(* CODESYS project SPT_XPlanar.library
   Company: Beckhoff Automation LLC
   DefaultNamespace: SPT_XPlanar
   Version: 3.2.0
   Placeholder: SPT_XPlanar
   Title: SPT_XPlanar

Project tree, tasks and I/O mapping:
  libraries: SPT Base Types, * (Beckhoff Automation LLC); SPT Event Logger, * (Beckhoff Automation LLC); SPT Tracing, * (Beckhoff Automation LLC); SPT Utilities, * (Beckhoff Automation LLC); Tc2_Math, * (Beckhoff Automation GmbH); Tc2_Standard, * (Beckhoff Automation GmbH); Tc2_System, * (Beckhoff Automation GmbH); Tc2_Utilities, * (Beckhoff Automation GmbH); Tc3_EventLogger, * (Beckhoff Automation GmbH); Tc3_Mc3PlanarMotion, * (Beckhoff Automation GmbH); Tc3_Module, * (Beckhoff Automation GmbH); Tc3_Physics, * (Beckhoff Automation GmbH); Tc3_XPlanarStandard, * (Beckhoff Automation GmbH); Tc3_XPlanarUtility, * (Beckhoff Automation GmbH & Co. KG)
  DUT/
    HMI/
      data type ST_Xplanar_Command
      data type ST_Xplanar_Config
      data type ST_Xplanar_HMI
      data type ST_Xplanar_Status
  Mover/
    DUTs/
      HMI/
        data type ST_Mover_HMI
        data type ST_MoverCommand_HMI
        data type ST_MoverConfig_HMI
        data type ST_MoverStatus_HMI
      data type ST_MoveDynamics
    function block FB_XPlanarMover [ST]: ClearCmd, Destination, Error, ErrorID, ErrorInfo, InStation, MoveDynamics, MoverBTN, MoverIndex, MoverType, std, TrackId, Disable, Enable, FreeMove, Index, JoinTrack, LeaveTrack, Reset, SendToStation, Spin, SquareUp, Tilt, VerticalMove, ClearCmdError, CyclicLogic, HMICommunication, IODriver
    interface I_XPlanarMover: ClearCmd, FreeMove, Index, JoinTrack, LeaveTrack, SendToStation, Spin, SquareUp, Tilt, VerticalMove, Destination, Error, ErrorID, ErrorInfo, InStation, MoveDynamics, MoverBTN, MoverIndex, MoverType, std, TrackId
  Project Information/
    function F_GetCompany [ST]
    function F_GetTitle [ST]
    function F_GetVersion [ST]
  Station/
    DUT/
      HMI/
        data type ST_Station_HMI
        data type ST_StationCommand_HMI
        data type ST_StationConfig_HMI
        data type ST_StationStatus_HMI
      data type E_StationType
      data type E_XplanarStationState
    function block FB_MoverQueue [ST]: Clear, Count, Dequeue, Enqueue, FirstMover, LastMover, MoverIDs, Queue
    function block FB_XPlanarStationBase [ST]: CyclicLogic, HMICommunication, AllowQueing, CanReleaseMover, CurrentMover, Error, Execute, HasMover, ID, MoverQueue, NextStation, NumMoversRequired, Position, Recover, Reset, Size, StationComplete, StationReady, StationType, TrackID
    interface I_XPlanarStation: AllowQueing, CanReleaseMover, CurrentMover, Execute, HasMover, ID, MoverQueue, NextStation, NumMoversRequired, Position, Recover, Reset, Size, StationComplete, StationReady, StationType, TrackID
    global variables StationParameters
  Track/
    DUT/
      HMI/
        data type ST_Track_HMI
        data type ST_TrackCommand_HMI
        data type ST_TrackConfig_HMI
        data type ST_TrackStatus_HMI
    function block FB_XPlanarTrackSegment [ST]: Clear, Error, ErrorInfo, ID, MoverCount, OpMode, std, TrackLength, TrackTable, Build, CyclicLogic, HMICommunication
    interface I_XPlanarTrack: Clear, Error, ErrorInfo, ID, MoverCount, OpMode, std, TrackLength, TrackTable
  Version/
    global variables Global_Version
  function block FB_Component_XPlanar [ST]: CreateEvents, HMICommunication, Monitoring, CyclicLogic, Abort, BuildTracks, CheckMovers, CheckTilePower, EnableGroup, EnableMovers, EnableTracks, Initialize, MoverRedetect, RecoverStations, Reset, TileCount, TracksInitialized, Xpu
  global variables ip
  00000000-0000-0000-0000-000000000000|LICENSE
  LICENSE
*)

// DUT/HMI/ST_Xplanar_Command
TYPE ST_Xplanar_Command :
	STRUCT
	END_STRUCT
END_TYPE

// DUT/HMI/ST_Xplanar_Config
TYPE ST_Xplanar_Config :
	STRUCT
	END_STRUCT
END_TYPE

// DUT/HMI/ST_Xplanar_HMI
TYPE ST_Xplanar_HMI :
	STRUCT
		Config	: ST_Xplanar_Config;
		Command : ST_Xplanar_Command;
		Status	: ST_Xplanar_Status;
	END_STRUCT
END_TYPE

// DUT/HMI/ST_Xplanar_Status
TYPE ST_Xplanar_Status :
	STRUCT
		Initialized		 : BOOL;
		TileCount		 : UDINT;
		NumberOfMovers	 : UDINT;
		NumberOfTracks	 : UDINT;
		NumberOfStations : UDINT;
		PowerOK			 : BOOL;
	END_STRUCT
END_TYPE

// Mover/DUTs/HMI/ST_Mover_HMI
TYPE ST_Mover_HMI :
	STRUCT
		Command : ST_MoverCommand_HMI;
		Config	: ST_MoverConfig_HMI;
		Status	: ST_MoverStatus_HMI;
	END_STRUCT
END_TYPE

// Mover/DUTs/HMI/ST_MoverCommand_HMI
TYPE ST_MoverCommand_HMI :
	STRUCT
	END_STRUCT
END_TYPE

// Mover/DUTs/HMI/ST_MoverConfig_HMI
TYPE ST_MoverConfig_HMI :
	STRUCT
	END_STRUCT
END_TYPE

// Mover/DUTs/HMI/ST_MoverStatus_HMI
TYPE ST_MoverStatus_HMI :
	STRUCT
		Enabled		: BOOL;
		Busy		: BOOL;
		Error		: BOOL;
		ID			: STRING(13);
		CommandMode : MC_PLANAR_MOVER_COMMAND_MODE;
		TrackID		: UDINT;
	END_STRUCT
END_TYPE

// Mover/DUTs/ST_MoveDynamics
TYPE ST_MoveDynamics :
	STRUCT
		VeloSlow : LREAL := 150;
		Velo	 : LREAL := 400;
		Accel	 : LREAL := 2000;
		Decel	 : LREAL := 2000;
		Jerk	 : LREAL := 20000;
		VeloRot	 : LREAL := 400.0;
		AccelRot : LREAL := 16000.0;
		JerkRot	 : LREAL := 100000.0;
		Gap		 : LREAL := 300.0;
	END_STRUCT
END_TYPE

// Station/DUT/HMI/ST_Station_HMI
TYPE ST_Station_HMI :
	STRUCT
		Config	: ST_StationConfig_HMI;
		Command : ST_StationCommand_HMI;
		Status	: ST_StationStatus_HMI;
	END_STRUCT
END_TYPE

// Station/DUT/HMI/ST_StationCommand_HMI
TYPE ST_StationCommand_HMI :
	STRUCT
	END_STRUCT
END_TYPE

// Station/DUT/HMI/ST_StationConfig_HMI
TYPE ST_StationConfig_HMI :
	STRUCT
	END_STRUCT
END_TYPE

// Station/DUT/HMI/ST_StationStatus_HMI
TYPE ST_StationStatus_HMI :
	STRUCT
		HasMover : BOOL;
		MoverID	 : STRING(13);
	END_STRUCT
END_TYPE

// Station/DUT/E_StationType
{attribute 'qualified_only'}
TYPE E_StationType : (
		Process		  := 0,
		DecisionPoint := 1,
		MultiMover	  := 2
	) UDINT;
END_TYPE

// Station/DUT/E_XplanarStationState
{attribute 'qualified_only'}
{attribute 'strict'}
TYPE E_XplanarStationState : (
		StationIdle := 0,
		ProcessMover,
		SquareUpMover,
		SendMoverAway,
		CycleComplete,
		SendQueue,
		StationError
	);
END_TYPE

// Track/DUT/HMI/ST_Track_HMI
TYPE ST_Track_HMI :
	STRUCT
		Config	: ST_TrackConfig_HMI;
		Command : ST_TrackCommand_HMI;
		Status	: ST_TrackStatus_HMI;
	END_STRUCT
END_TYPE

// Track/DUT/HMI/ST_TrackCommand_HMI
TYPE ST_TrackCommand_HMI :
	STRUCT
	END_STRUCT
END_TYPE

// Track/DUT/HMI/ST_TrackConfig_HMI
TYPE ST_TrackConfig_HMI :
	STRUCT
	END_STRUCT
END_TYPE

// Track/DUT/HMI/ST_TrackStatus_HMI
TYPE ST_TrackStatus_HMI :
	STRUCT
		State			 : MC_PLANAR_STATE;
		OperationMode	 : MC_PLANAR_TRACK_OPERATION_MODE;
		MoverCount		 : UDINT;
		CalculatedLength : LREAL;
	END_STRUCT
END_TYPE

// Station/StationParameters
{attribute 'qualified_only'}
VAR_GLOBAL CONSTANT
	MaxMoversPerStation			: UDINT := 4;
END_VAR

// Version/Global_Version
{attribute 'TcGenerated'}
{attribute 'no-analysis'}
{attribute 'linkalways'}
// This function has been automatically generated from the project information.
VAR_GLOBAL CONSTANT
	{attribute 'const_non_replaced'}
	stLibVersion_SPT_XPlanar : ST_LibVersion := (iMajor := 3, iMinor := 2, iBuild := 0, iRevision := 0, nFlags := 1, sVersion := '3.2.0');
END_VAR

// ip
{attribute 'qualified_only'}
VAR_GLOBAL
	Movers	 : ARRAY[0..Tc3_XPlanarStandard.Params_XPlanar.moverCount] OF I_XPlanarMover;
	Tracks	 : ARRAY[0..Tc3_XPlanarStandard.Params_XPlanar.maxTrackCount] OF I_XPlanarTrack;
	Stations : ARRAY[0..Tc3_XPlanarStandard.Params_XPlanar.maxNumStation] OF I_XPlanarStation;
END_VAR

// Mover/FB_XPlanarMover
FUNCTION_BLOCK FB_XPlanarMover IMPLEMENTS I_XPlanarMover
VAR_INPUT
END_VAR

VAR_OUTPUT
END_VAR

VAR
	_Mover			  : FB_XPlanarMoverStandard;
	_MoverIndex		  : UDINT;
	_TrackId		  : UDINT;
	_MoverBTN		  : STRING[13];
	_MoverType		  : MoverType;
	_InStation		  : BOOL;
	ipDestination	  : I_XPlanarStation;
	ipIoDriver		  : I_TcIoXPlanarMover;
	_MoveDynamics	  : ST_MoveDynamics;
	_Error			  : BOOL;
	_ErrorID		  : UDINT;
	_ErrorInfo		  : STRING;
	LeaveTrackOptions : ST_LeaveTrackOptions;
	JoinTrackOptions  : ST_JoinTrackOptions;
	RotateOptions	  : ST_MoveCOptions;
	RotateDirection	  : Tc3_Mc3PlanarMotion.MC_DIRECTION;
	CommandState	  : (Init,
		Command,
		Feedback,
		Complete,
		CmdError);
	Mover_HMI		 : ST_Mover_HMI;
	ClosestSquarePos : LREAL;
END_VAR

METHOD ClearCmd : BOOL
VAR_INPUT
END_VAR
CommandState := Init;
ClearCmdError();
ClearCmd := true;
END_METHOD

PROPERTY Destination : I_XPlanarStation
GET
Destination := ipDestination;
END_GET
SET
ipDestination := Destination;
END_SET
END_PROPERTY

PROPERTY Error : BOOL
GET
END_GET
END_PROPERTY

PROPERTY ErrorID : UDINT
GET
END_GET
END_PROPERTY

PROPERTY ErrorInfo : STRING
GET
END_GET
END_PROPERTY

PROPERTY InStation : BOOL
GET
InStation := _InStation;
END_GET
SET
_InStation := InStation;
END_SET
END_PROPERTY

PROPERTY MoveDynamics : REFERENCE TO ST_MoveDynamics
GET
MoveDynamics ref= _MoveDynamics;
END_GET
END_PROPERTY

PROPERTY MoverBTN : STRING
GET
MoverBTN := _MoverBTN;
END_GET
SET
_MoverBTN := MoverBTN;
END_SET
END_PROPERTY

PROPERTY MoverIndex : UDINT
GET
MoverIndex := _MoverIndex;
END_GET
SET
_MoverIndex := MoverIndex;
END_SET
END_PROPERTY

PROPERTY MoverType : MoverType
GET
MoverType := _MoverType;
END_GET
SET
_MoverType := MoverType;
END_SET
END_PROPERTY

PROPERTY std : I_XPlanarMoverStandard
GET
std := _Mover;
END_GET
END_PROPERTY

PROPERTY TrackId : UDINT
GET
TrackId := _TrackId;
END_GET
SET
_TrackId := TrackId;
END_SET
END_PROPERTY

METHOD Disable : BOOL
VAR
	Result : BOOL;
END_VAR
Disable := FALSE;
CASE CommandState OF
	Init:
		ClearCmdError();
		IF _Mover.P_State = MC_PLANAR_STATE.Disabled THEN
			CommandState := Complete;
		ELSE
			CommandState := Command;
		END_IF

	Command:
		Result		 := _Mover.Disable('Disable');
		CommandState := Feedback;

	Feedback:
		IF _Mover.P_Disable.Done OR _Mover.P_State = MC_PLANAR_STATE.Disabled THEN
			CommandState := Complete;
		ELSIF _Mover.P_Disable.Error THEN
			CommandState := CmdError;
		END_IF

	Complete:
		Disable		 := TRUE;
		CommandState := Init;

	CmdError:
		_Error		 := TRUE;
		_ErrorID	 := _Mover.P_Disable.ErrorID;
		_ErrorInfo	 := 'MoverDisableError';
		Disable		 := TRUE;
		CommandState := Init;
END_CASE
END_METHOD

METHOD Enable : BOOL
VAR
	Result : BOOL;
END_VAR
Enable := FALSE;
CASE CommandState OF
	Init:
		ClearCmdError();
		IF ipIoDriver <> 0 THEN
			_MoverBTN  := ipIoDriver.GetBtn();
			_MoverType := ipIoDriver.GetMoverType();
		END_IF

		IF _Mover.P_State = MC_PLANAR_STATE.Enabled THEN
			CommandState := Complete;
		ELSE
			CommandState := Command;
		END_IF

	Command:
		Result		 := _Mover.Enable('Enable');
		CommandState := Feedback;

	Feedback:
		IF _Mover.P_Enable.Done OR _Mover.P_State = MC_PLANAR_STATE.Enabled THEN
			CommandState := Complete;
		ELSIF _Mover.P_Enable.Error THEN
			CommandState := CmdError;
		END_IF

	Complete:
		Enable		 := TRUE;
		CommandState := Init;

	CmdError:
		_Error		 := TRUE;
		_ErrorID	 := _Mover.P_Enable.ErrorID;
		_ErrorInfo	 := 'MoverEnableError';
		CommandState := Init;
END_CASE
END_METHOD

METHOD FreeMove : BOOL
VAR_INPUT
	XPosition : LREAL;
	YPosition : LREAL;
END_VAR

VAR_INST
	Position : PositionXYC;
END_VAR

VAR
	Result : BOOL;
END_VAR
FreeMove := FALSE;
CASE CommandState OF
	Init:
		ClearCmdError();
		CommandState := Command;

	Command:
		Position.SetValuesXYC(XPosition, YPosition, 0.0);
		Result := _Mover.MoveToPosition(CONCAT(CONCAT('MoveTo ', TO_STRING(XPosition)), CONCAT(', ', TO_STRING(YPosition))),
										Position,
										_MoveDynamics.Velo,
										_MoveDynamics.Accel,
										_MoveDynamics.Decel,
										_MoveDynamics.Jerk);

		CommandState := Feedback;

	Feedback:
		IF _Mover.P_MoveToPosition.Done THEN
			CommandState := Complete;
		ELSIF _Mover.P_MoveToPosition.Error THEN
			CommandState := CmdError;
		END_IF

	Complete:
		FreeMove	 := TRUE;
		CommandState := Init;

	CmdError:
		FreeMove	 := TRUE;
		CommandState := Init;
		_Error		 := TRUE;
		_ErrorID	 := _Mover.P_MoveToPosition.ErrorID;
		_ErrorInfo	 := 'MoveToPositionError';
END_CASE
END_METHOD

{attribute 'TcRpcEnable'}
METHOD Index : BOOL
VAR_INPUT
	Distance : LREAL;
END_VAR

VAR
	Result : BOOL;
END_VAR
Index := FALSE;
CASE CommandState OF
	Init:
		ClearCmdError();
		CommandState := Command;

	Command:
		IF Distance < 0 THEN
			RotateDirection := Tc3_Mc3PlanarMotion.MC_DIRECTION.mcDirectionNegative;
		ELSE
			RotateDirection := Tc3_Mc3PlanarMotion.MC_DIRECTION.mcDirectionPositive;
		END_IF
		
		RotateOptions.additionalTurns := 0;
		RotateOptions.direction		  := RotateDirection;
		Result						  := _Mover.MoveC(CONCAT('Index ', TO_STRING(Distance)),
													  ABS(Distance),
													  _MoveDynamics.VeloRot,
													  _MoveDynamics.AccelRot,
													  _MoveDynamics.AccelRot,
													  _MoveDynamics.JerkRot,
													  RotateOptions);

		CommandState := Feedback;

	Feedback:
		IF _Mover.P_MoveC.Done THEN
			CommandState := Complete;
		ELSIF _Mover.P_MoveC.Error THEN
			CommandState := CmdError;
		END_IF

	Complete:
		Index		 := TRUE;
		CommandState := Init;

	CmdError:
		Index		 := TRUE;
		CommandState := Init;
		_Error		 := TRUE;
		_ErrorID	 := _Mover.P_MoveC.ErrorID;
		_ErrorInfo	 := 'MoverCError';
END_CASE
END_METHOD

{attribute 'TcRpcEnable'}
METHOD JoinTrack : BOOL
VAR_INPUT
	ipTrack : I_XPlanarTrack;
END_VAR

VAR
	Result : BOOL;
END_VAR
JoinTrack := FALSE;
IF ipTrack <> 0 THEN
	CASE CommandState OF
		Init:
			ClearCmdError();
			CommandState := Command;

		Command:
			IF ipTrack.ID <> 0 THEN
				JoinTrackOptions.useOrientation := FALSE;
				Result							:= _Mover.JoinTrack(CONCAT('JoinTrack ', TO_STRING(ipTrack.ID)),
																	ipTrack.std,
																	_MoveDynamics.VeloSlow,
																	_MoveDynamics.Accel,
																	_MoveDynamics.Jerk,
																	JoinTrackOptions);

				CommandState := Feedback;
			ELSE
				; ///Marc TODO: // HOw to handle
			END_IF

		Feedback:
			IF _Mover.P_JoinTrack.Done THEN
				CommandState := Complete;
			ELSIF _Mover.P_JoinTrack.Error THEN
				CommandState := CmdError;
			END_IF

		Complete:
			JoinTrack	 := TRUE;
			CommandState := Init;

		CmdError:
			JoinTrack	 := TRUE;
			CommandState := Init;
			_Error		 := TRUE;
			_ErrorID	 := _Mover.P_JoinTrack.ErrorID;
			_ErrorInfo	 := 'JoinTrackError';
	END_CASE
ELSE
	; ///Marc TODO: how to handle
END_IF
END_METHOD

{attribute 'TcRpcEnable'}
METHOD LeaveTrack : BOOL
VAR_INPUT
	DestinationX : LREAL;
	DestinationY : LREAL;
END_VAR

VAR_INST
	Destination : PositionXYC;
END_VAR

VAR
	Result : BOOL;
END_VAR
LeaveTrack := FALSE;
CASE CommandState OF
	Init:
		ClearCmdError();
		Destination.SetValuesXYC(DestinationX, DestinationY, 0.0);
		CommandState := Command;

	Command:
		RotateOptions.additionalTurns := 0;
		RotateOptions.direction		  := Tc3_Mc3PlanarMotion.MC_DIRECTION.mcDirectionPositive;
		Result						  := _Mover.LeaveTrack('LeaveTrack',
														   Destination,
														   _MoveDynamics.VeloSlow,
														   _MoveDynamics.Accel,
														   _MoveDynamics.Decel,
														   _MoveDynamics.Jerk,
														   LeaveTrackOptions);

		CommandState := Feedback;

	Feedback:
		IF _Mover.P_LeaveTrack.Done THEN
			CommandState := Complete;
		ELSIF _Mover.P_LeaveTrack.Error THEN
			CommandState := CmdError;
		END_IF

	Complete:
		LeaveTrack	 := TRUE;
		CommandState := Init;

	CmdError:
		LeaveTrack	 := TRUE;
		CommandState := Init;
		_Error		 := TRUE;
		_ErrorID	 := _Mover.P_LeaveTrack.ErrorID;
		_ErrorInfo	 := 'LeaveTrackError';
END_CASE
END_METHOD

//! @summary Clears error flags and error IDs for this component
METHOD PUBLIC Reset : BOOL
VAR
	Result : BOOL;
END_VAR
Reset := FALSE;
CASE CommandState OF
	Init:
		_Error	 := FALSE;
		_ErrorID := 0;
		IF _Mover.P_State <> MC_PLANAR_STATE.Error THEN
			CommandState := Complete;
		ELSE
			CommandState := Command;
		END_IF

		CommandState := Command;

	Command:
		Result		 := _Mover.Reset('Reset');
		CommandState := Feedback;

	Feedback:
		IF _Mover.P_Reset.Done OR _Mover.P_State <> MC_PLANAR_STATE.Error THEN
			CommandState := Complete;
		ELSIF _Mover.P_Enable.Error THEN
			CommandState := CmdError;
		END_IF

	Complete:
		Reset		 := TRUE;
		CommandState := Init;

	CmdError:
		_Error		 := TRUE;
		_ErrorID	 := _Mover.P_Reset.ErrorID;
		_ErrorInfo	 := 'MoverResetError';
		Reset		 := TRUE;
		CommandState := Init;
END_CASE
END_METHOD

{attribute 'TcRpcEnable'}
METHOD SendToStation : BOOL
VAR_INPUT
	ipDestinationLocal : I_XPlanarStation; (*///Marc TODO:  the FB_Mover has a ipDestination.  
									///Does this mehtod want to use the one passed here?  
									So I added the Local to the name as to not be confused with the FB one*)
END_VAR

VAR_INST
	CorrectedPos : PositionXYC;
	OnTrackPos	 : LREAL;
END_VAR

VAR
	Result : BOOL;
END_VAR
SendToStation := FALSE;
IF ipDestinationLocal <> 0 THEN
	CASE CommandState OF
		Init:
			ClearCmdError();
			CommandState := Command;

		Command:
			ipDestination := ipDestinationLocal;
			IF _Mover.P_CommandMode = MC_PLANAR_MOVER_COMMAND_MODE.OnTrack THEN
				IF ipDestinationLocal.TrackID <> 0 THEN
					IF ipDestinationLocal.TrackID.std <> 0 THEN
						OnTrackPos := ipDestinationLocal.TrackID.std.GetTrackPositionAt(ipDestinationLocal.Position);
						Result	   := _Mover.MoveOnTrack(CONCAT('SendToStation ', TO_STRING(ipDestinationLocal.ID)),
														 ipDestinationLocal.TrackID.std,
														 OnTrackPos,
														 _MoveDynamics.Velo,
														 _MoveDynamics.Accel,
														 _MoveDynamics.Jerk,
														 _MoveDynamics.Gap,
														 Tc3_Mc3PlanarMotion.MC_DIRECTION.mcDirectionPositive);
					ELSE
						; /// Marc TODO:  how to handle std null
					END_IF
				END_IF
			ELSIF _Mover.P_CommandMode = MC_PLANAR_MOVER_COMMAND_MODE.FreeMovement THEN
				CorrectedPos.SetValuesXYC(ipDestinationLocal.Position.x, ipDestinationLocal.Position.y, _Mover.P_ClosestQuaterAngle);
				Result := _Mover.MoveToPosition(CONCAT('SendToStation ', TO_STRING(ipDestinationLocal.ID)),
												CorrectedPos,
												_MoveDynamics.Velo,
												_MoveDynamics.Accel,
												_MoveDynamics.Decel,
												_MoveDynamics.Jerk);
			END_IF

			CommandState := Feedback;

		Feedback:
			IF _Mover.P_CommandMode = MC_PLANAR_MOVER_COMMAND_MODE.OnTrack THEN
				IF _Mover.P_MoveOnTrack.Active OR _Mover.P_MoveOnTrack.Done THEN
					CommandState := Complete;
				ELSIF _Mover.P_MoveOnTrack.Error THEN
					CommandState := CmdError;
				END_IF
			ELSIF _Mover.P_CommandMode = MC_PLANAR_MOVER_COMMAND_MODE.FreeMovement THEN
				IF _Mover.P_MoveToPosition.Active OR _Mover.P_MoveToPosition.Done THEN
					CommandState := Complete;
				ELSIF _Mover.P_MoveToPosition.Error THEN
					CommandState := CmdError;
				END_IF
			END_IF

		Complete:
			SendToStation := TRUE;
			CommandState  := Init;

		CmdError:
			SendToStation := TRUE;
			CommandState  := Init;
			_Error		  := TRUE;
			IF _Mover.P_CommandMode = MC_PLANAR_MOVER_COMMAND_MODE.OnTrack THEN
				_ErrorID   := _Mover.P_MoveOnTrack.ErrorID;
				_ErrorInfo := 'MoverOnTrackError';
			ELSIF _Mover.P_CommandMode = MC_PLANAR_MOVER_COMMAND_MODE.FreeMovement THEN
				_ErrorID   := _Mover.P_MoveToPosition.ErrorID;
				_ErrorInfo := 'MoverToPositionError';
			END_IF
	END_CASE
ELSE
	; ///Marc TODO: how to handle this?	
END_IF
END_METHOD

{attribute 'TcRpcEnable'}
METHOD Spin : BOOL
VAR_INPUT
	NumOfTurns : DINT;
END_VAR

VAR
	Result : BOOL;
END_VAR
Spin := FALSE;
CASE CommandState OF
	Init:
		ClearCmdError();	
		CommandState := Command;

	Command:
		IF NumOfTurns < 0 THEN
			RotateDirection := Tc3_Mc3PlanarMotion.MC_DIRECTION.mcDirectionNegative;
		ELSE
			RotateDirection := Tc3_Mc3PlanarMotion.MC_DIRECTION.mcDirectionPositive;
		END_IF
		
		RotateOptions.additionalTurns := ABS(NumOfTurns);
		RotateOptions.direction		  := RotateDirection;
		Result						  := _Mover.MoveC(CONCAT('Spin ', TO_STRING(NumOfTurns)),
													  0.0,
													  _MoveDynamics.VeloRot,
													  _MoveDynamics.AccelRot,
													  _MoveDynamics.AccelRot,
													  _MoveDynamics.JerkRot,
													  RotateOptions);

		CommandState := Feedback;

	Feedback:
		IF _Mover.P_MoveC.Done THEN
			CommandState := Complete;
		ELSIF _Mover.P_MoveC.Error THEN
			CommandState := CmdError;
		END_IF

	Complete:
		Spin		 := TRUE;
		CommandState := Init;

	CmdError:
		Spin		 := TRUE;
		CommandState := Init;
		_Error		 := TRUE;
		_ErrorID	 := _Mover.P_MoveC.ErrorID;
		_ErrorInfo	 := 'MoveCError';
END_CASE
END_METHOD

{attribute 'TcRpcEnable'}
METHOD SquareUp : BOOL
VAR
	Result : BOOL;
END_VAR
SquareUp := FALSE;
CASE CommandState OF
	Init:
		ClearCmdError();
		CommandState := Command;

	Command:
		RotateOptions.additionalTurns := 0;
		RotateOptions.direction		  := Tc3_Mc3PlanarMotion.MC_DIRECTION.mcDirectionShortestWay;
		Result						  := _Mover.MoveC('SquareMover',
													  ClosestSquarePos,
													  _MoveDynamics.VeloRot,
													  _MoveDynamics.AccelRot,
													  _MoveDynamics.AccelRot,
													  _MoveDynamics.JerkRot,
													  RotateOptions);

		CommandState := Feedback;

	Feedback:
		IF _Mover.P_MoveC.Done THEN
			SquareUp	 := TRUE;
			CommandState := Init;
		ELSIF _Mover.P_MoveC.Error THEN
			CommandState := CmdError;
		END_IF

	CmdError:
		_Error		 := TRUE;
		_ErrorID	 := _Mover.P_MoveC.ErrorID;
		_ErrorInfo	 := 'MoveCError';
		SquareUp	 := TRUE;
		CommandState := Init;
END_CASE
END_METHOD

{attribute 'TcRpcEnable'}
METHOD Tilt : BOOL
VAR_INPUT
	AxisAPosition : LREAL;
	AxisBPosition : LREAL;
END_VAR

VAR
	Result : BOOL;
END_VAR
Tilt := FALSE;
CASE CommandState OF
	Init:
		ClearCmdError();
		CommandState := Command;

	Command:
		Result := _Mover.MoveA(CONCAT('TiltMoveA ', TO_STRING(AxisAPosition)),
							   AxisAPosition,
							   _MoveDynamics.VeloSlow,
							   _MoveDynamics.Accel,
							   _MoveDynamics.Accel,
							   _MoveDynamics.Jerk);

		Result := _Mover.MoveB(CONCAT('TiltMoveA ', TO_STRING(AxisBPosition)),
							   AxisBPosition,
							   _MoveDynamics.VeloSlow,
							   _MoveDynamics.Accel,
							   _MoveDynamics.Accel,
							   _MoveDynamics.Jerk);

		CommandState := Feedback;

	Feedback:
		IF _Mover.P_MoveA.Done AND _Mover.P_MoveB.Done THEN
			Tilt		 := TRUE;
			CommandState := Init;
		ELSIF _Mover.P_MoveA.Error OR _Mover.P_MoveA.Error THEN
			CommandState := CmdError;
		END_IF

	CmdError:
		_Error := TRUE;
		IF _Mover.P_MoveA.Error THEN
			_ErrorID   := _Mover.P_MoveA.ErrorID;
			_ErrorInfo := 'MoveAError';
		ELSIF _Mover.P_MoveB.Error THEN
			_ErrorID   := _Mover.P_MoveB.ErrorID;
			_ErrorInfo := 'MoverBError';
		END_IF

		Tilt		 := TRUE;
		CommandState := Init;
END_CASE
END_METHOD

{attribute 'TcRpcEnable'}
METHOD VerticalMove : BOOL
VAR_INPUT
	Position : LREAL;
END_VAR

VAR
	Result : BOOL;
END_VAR
VerticalMove := FALSE;
CASE CommandState OF
	Init:
		ClearCmdError();
		CommandState := Command;

	Command:
		Result := _Mover.MoveZ(CONCAT('ZAxisMove ', TO_STRING(Position)),
							   Position,
							   _MoveDynamics.VeloSlow,
							   _MoveDynamics.Accel,
							   _MoveDynamics.Accel,
							   _MoveDynamics.Jerk);

		CommandState := Feedback;

	Feedback:
		IF _Mover.P_MoveZ.Done THEN
			VerticalMove := TRUE;
			CommandState := Init;
		ELSIF _Mover.P_MoveZ.Error THEN
			CommandState := CmdError;
		END_IF

	CmdError:
		VerticalMove := TRUE;
		CommandState := Init;
		_Error		 := TRUE;
		_ErrorID	 := _Mover.P_MoveZ.ErrorID;
		_ErrorInfo	 := 'MoveZError';
END_CASE
END_METHOD

METHOD PRIVATE ClearCmdError
VAR_INPUT
END_VAR
_Error	   := FALSE;
_ErrorID   := 0;
_ErrorInfo := '';
END_METHOD

//! @summary This method serves as the entry point for all underlying FB logic
METHOD PUBLIC CyclicLogic
//! @description This method should be called cyclically by descendant function blocks by invoking <c>SUPER^.CyclicLogic()</c>.  Alternatively, the contents of this method could be reimplemented entirely in which case a call to this method would not be necessary.
VAR
	Result : BOOL;
END_VAR
Result				 := _Mover.Cycle();								   //Keep the mover nc object alive
_Mover.P_SetPosition := _Mover.stMoverRef.MCTOPLC.SET.SetPos;		   //Update the Set position of MoverStandard
ClosestSquarePos	 := ABS(LMOD(_Mover.P_ClosestQuaterAngle, 360.0)); //Calculate the closest 'square position' for xy movement
HMICommunication();													   //Update mover status for HMI
END_METHOD

METHOD PROTECTED HMICommunication
VAR_INPUT
END_VAR
Mover_HMI.Status.Enabled	 := _Mover.P_State = MC_PLANAR_STATE.Enabled;
Mover_HMI.Status.Busy		 := _Mover.P_Busy; //Handle the Busy bit of the component
Mover_HMI.Status.Error		 := _Mover.P_State = MC_PLANAR_STATE.Error;
Mover_HMI.Status.ID			 := _MoverBTN;
Mover_HMI.Status.CommandMode := _Mover.P_CommandMode;
Mover_HMI.Status.TrackID	 := _Mover.P_TrackId;
END_METHOD

PROPERTY IODriver : I_TcIoXPlanarMover
SET
ipIoDriver := IoDriver;
END_SET
END_PROPERTY

END_FUNCTION_BLOCK

// Mover/I_XPlanarMover
INTERFACE I_XPlanarMover

METHOD ClearCmd : BOOL
VAR_INPUT
END_VAR
END_METHOD

METHOD FreeMove : BOOL
VAR_INPUT
	XPosition : LREAL;
	YPosition : LREAL;
END_VAR
END_METHOD

{attribute 'TcRpcEnable'}
METHOD Index : BOOL
VAR_INPUT
	Distance : LREAL;
END_VAR
END_METHOD

{attribute 'TcRpcEnable'}
METHOD JoinTrack : BOOL
VAR_INPUT
	ipTrack : I_XPlanarTrack;
END_VAR
END_METHOD

{attribute 'TcRpcEnable'}
METHOD LeaveTrack : BOOL
VAR_INPUT
	DestinationX : LREAL;
	DestinationY : LREAL;
END_VAR
END_METHOD

{attribute 'TcRpcEnable'}
METHOD SendToStation : BOOL
VAR_INPUT
	ipDestinationLocal : I_XPlanarStation;
END_VAR
END_METHOD

{attribute 'TcRpcEnable'}
METHOD Spin : BOOL
VAR_INPUT
	NumOfTurns : DINT;
END_VAR
END_METHOD

{attribute 'TcRpcEnable'}
METHOD SquareUp : BOOL
END_METHOD

{attribute 'TcRpcEnable'}
METHOD Tilt : BOOL
VAR_INPUT
	AxisAPosition : LREAL;
	AxisBPosition : LREAL;
END_VAR
END_METHOD

{attribute 'TcRpcEnable'}
METHOD VerticalMove : BOOL
VAR_INPUT
	Position : LREAL;
END_VAR
END_METHOD

PROPERTY Destination : I_XPlanarStation
GET
END_GET
SET
END_SET
END_PROPERTY

PROPERTY Error : BOOL
GET
END_GET
END_PROPERTY

PROPERTY ErrorID : UDINT
GET
END_GET
END_PROPERTY

PROPERTY ErrorInfo : STRING
GET
END_GET
END_PROPERTY

PROPERTY InStation : BOOL
GET
END_GET
SET
END_SET
END_PROPERTY

PROPERTY MoveDynamics : REFERENCE TO ST_MoveDynamics
GET
END_GET
END_PROPERTY

PROPERTY MoverBTN : STRING
GET
END_GET
SET
END_SET
END_PROPERTY

PROPERTY MoverIndex : UDINT
GET
END_GET
SET
END_SET
END_PROPERTY

PROPERTY MoverType : MoverType
GET
END_GET
SET
END_SET
END_PROPERTY

PROPERTY std : I_XPlanarMoverStandard
GET
END_GET
END_PROPERTY

PROPERTY TrackId : UDINT
GET
END_GET
SET
END_SET
END_PROPERTY

END_INTERFACE

// Track/I_XPlanarTrack
INTERFACE I_XPlanarTrack

METHOD Clear : BOOL
END_METHOD

PROPERTY Error : BOOL
GET
END_GET
END_PROPERTY

PROPERTY ErrorInfo : STRING
GET
END_GET
END_PROPERTY

PROPERTY ID : UDINT
GET
END_GET
SET
END_SET
END_PROPERTY

PROPERTY MoverCount : UDINT
GET
END_GET
END_PROPERTY

PROPERTY OpMode : MC_PLANAR_TRACK_OPERATION_MODE
GET
END_GET
END_PROPERTY

PROPERTY std : I_TrackStandard
GET
END_GET
END_PROPERTY

PROPERTY TrackLength : LREAL
GET
END_GET
END_PROPERTY

PROPERTY TrackTable : REFERENCE TO FB_TrackTable
GET
END_GET
END_PROPERTY

END_INTERFACE

// Station/I_XPlanarStation
INTERFACE I_XPlanarStation

PROPERTY AllowQueing : BOOL
GET
END_GET
SET
END_SET
END_PROPERTY

PROPERTY CanReleaseMover : BOOL
SET
END_SET
END_PROPERTY

PROPERTY CurrentMover : I_XPlanarMover
GET
END_GET
END_PROPERTY

METHOD Execute
END_METHOD

PROPERTY HasMover : BOOL
GET
END_GET
SET
END_SET
END_PROPERTY

PROPERTY ID : UDINT
GET
END_GET
SET
END_SET
END_PROPERTY

PROPERTY MoverQueue : REFERENCE TO FB_MoverQueue
GET
END_GET
END_PROPERTY

PROPERTY NextStation : I_XPlanarStation
GET
END_GET
SET
END_SET
END_PROPERTY

PROPERTY NumMoversRequired : UDINT
GET
END_GET
SET
END_SET
END_PROPERTY

PROPERTY Position : REFERENCE TO PositionXYC
GET
END_GET
END_PROPERTY

METHOD Recover : BOOL
END_METHOD

METHOD Reset : BOOL
END_METHOD

PROPERTY Size : REFERENCE TO Position2D_LREAL
GET
END_GET
END_PROPERTY

PROPERTY StationComplete : BOOL
SET
END_SET
END_PROPERTY

PROPERTY StationReady : BOOL
GET
END_GET
END_PROPERTY

PROPERTY StationType : E_StationType
GET
END_GET
SET
END_SET
END_PROPERTY

PROPERTY TrackID : I_XPlanarTrack
GET
END_GET
SET
END_SET
END_PROPERTY

END_INTERFACE

// Station/FB_MoverQueue
//=============================================================================

//	FB_MoverQueue

//=============================================================================

//

//	FIFO Queue for use by stations

//

//-----------------------------------------------------------------------------
FUNCTION_BLOCK FB_MoverQueue
VAR
	MoversInQueue : UDINT := 0;
	ipMovers	  : ARRAY[1..StationParameters.MaxMoversPerStation] OF I_XPlanarMover;
END_VAR

//=============================================================================

//	Method Clear()

//=============================================================================

//

//	Brute force reset of buffer

//

//-----------------------------------------------------------------------------
METHOD Clear : BOOL
MEMSET(ADR(ipMovers), 0, SIZEOF(ipMovers));
MoversInQueue := 0;
Clear		  := TRUE;
END_METHOD

PROPERTY Count : UDINT
GET
VAR
	i	 : UDINT;
	temp : UDINT;
END_VAR
Count := MoversInQueue;
END_GET
END_PROPERTY

METHOD Dequeue : BOOL
IF MoversInQueue > 0 THEN
	ipMovers[1].InStation := FALSE;
	MEMSET(ADR(ipMovers[1]), 0, SIZEOF(ipMovers[1]));
	MoversInQueue := MoversInQueue - 1;
	IF MoversInQueue > 0 THEN
		MEMMOVE(ADR(ipMovers[1]), ADR(ipMovers[2]), SIZEOF(ipMovers[2]) * MoversInQueue);
		MEMSET(ADR(ipMovers[MoversInQueue + 1]), 0, (SIZEOF(ipMovers[1]) * (StationParameters.MaxMoversPerStation - MoversInQueue)));
	END_IF

	Dequeue := TRUE;
END_IF
END_METHOD

METHOD Enqueue : BOOL
VAR_INPUT
	ipMover : I_XPlanarMover;
END_VAR
IF MoversInQueue < StationParameters.MaxMoversPerStation THEN
	MoversInQueue			:= MoversInQueue + 1;
	ipMover.InStation		:= TRUE;
	ipMovers[MoversInQueue] := ipMover;
	Enqueue					:= TRUE;
END_IF
END_METHOD

PROPERTY FirstMover : I_XPlanarMover
GET
IF MoversInQueue > 0 THEN
	FirstMover := ipMovers[1];
END_IF
END_GET
END_PROPERTY

PROPERTY LastMover : I_XPlanarMover
GET
IF MoversInQueue > 0 THEN
	LastMover := ipMovers[MoversInQueue];
END_IF
END_GET
END_PROPERTY

PROPERTY MoverIDs : ARRAY[1..StationParameters.MaxMoversPerStation] OF UDINT
GET
VAR
	i : UDINT;
END_VAR
FOR i := 1 TO MoversInQueue DO
	IF ipMovers[i] <> 0 THEN
		MoverIDs[i] := ipMovers[i].MoverIndex;
	END_IF
END_FOR
END_GET
END_PROPERTY

PROPERTY Queue : REFERENCE TO ARRAY[1..StationParameters.MaxMoversPerStation] OF I_XPlanarMover;
GET
VAR
	i : UDINT;
END_VAR
Queue ref= ipMovers;
END_GET
END_PROPERTY

END_FUNCTION_BLOCK

// Project Information/F_GetCompany
// This function has been automatically generated from the project information.
{attribute 'signature_flag' := '1073741824'}
{attribute 'TcGenerated'}
{attribute 'no-analysis'}
FUNCTION F_GetCompany : WSTRING
VAR_INPUT
	
END_VAR

F_GetCompany := "Beckhoff Automation LLC";

END_FUNCTION

// Project Information/F_GetTitle
// This function has been automatically generated from the project information.
{attribute 'signature_flag' := '1073741824'}
{attribute 'TcGenerated'}
{attribute 'no-analysis'}
FUNCTION F_GetTitle : WSTRING
VAR_INPUT
	
END_VAR

F_GetTitle := "SPT_XPlanar";

END_FUNCTION

// Project Information/F_GetVersion
// This function has been automatically generated from the project information.
{attribute 'signature_flag' := '1073741824'}
{attribute 'TcGenerated'}
{attribute 'no-analysis'}
FUNCTION F_GetVersion : ST_LibVersion
VAR_INPUT
	
END_VAR

F_GetVersion.iMajor := 3;
F_GetVersion.iMinor := 2;
F_GetVersion.iBuild := 0;
F_GetVersion.iRevision := 0;
F_GetVersion.sVersion := '3.2.0';
F_GetVersion.nFlags := 1;

END_FUNCTION

// Station/FB_XPlanarStationBase
FUNCTION_BLOCK FB_XPlanarStationBase EXTENDS FB_ComponentBase IMPLEMENTS I_XPlanarStation
VAR
	_Position			 : PositionXYC; //Position of center of the zone
	ipCurrentMover		 : I_XPlanarMover;
	_MoverQueue			 : FB_MoverQueue;
	_NumMoversRequired	 : UDINT := 1;
	_ID					 : UDINT;
	_Size				 : Position2D_LREAL := (x := 120, y := 120); //Size of zone in mm
	_HasMover			 : BOOL;
	ipTrackID			 : I_XPlanarTrack; //ID of track that zone resides on
	_CanReleaseMover	 : BOOL := TRUE;   //Set to 0 if station area is blocked
	_StationReady AT %Q* : BOOL;
	ipNextStation		 : I_XPlanarStation;
	_AllowQueing		 : BOOL := TRUE;
	_StationComplete	 : BOOL;
	_StationType		 : E_StationType := E_StationType.Process;
	ipMovers			 : REFERENCE TO ARRAY[1..Tc3_XPlanarStandard.Params_XPlanar.moverCount] OF I_XPlanarMover;
	PrepState			 : UDINT;
	Station_HMI			 : ST_Station_HMI;
	StationState		 : E_XplanarStationState;
END_VAR

METHOD CyclicLogic
VAR_INST
	idx : UDINT;
END_VAR
FOR idx := 1 TO Tc3_XPlanarStandard.Params_XPlanar.moverCount DO
	IF ip.Movers[idx] <> 0 THEN
		IF _Position.x > 0 AND _Position.y > 0 THEN
			IF (ip.Movers[idx].std.P_ActPosition.x + 50 >= _Position.x - (_Size.x / 2) AND ip.Movers[idx].std.P_ActPosition.x - 50 <= _Position.x + (_Size.x / 2)) AND
			   (ip.Movers[idx].std.P_ActPosition.y + 50 >= _Position.y - (_Size.y / 2) AND ip.Movers[idx].std.P_ActPosition.y - 50 <= _Position.y + (_Size.y / 2)) THEN
				IF ip.Movers[idx].Destination <> 0 THEN
					IF ip.Movers[idx].Destination.ID = _ID AND NOT ip.Movers[idx].InStation THEN
						_MoverQueue.Enqueue(ip.Movers[idx]);
					END_IF
				END_IF
			END_IF
		END_IF
	END_IF
END_FOR

IF _MoverQueue.Count > 0 THEN
	_HasMover := TRUE;
	ipCurrentMover := _MoverQueue.FirstMover;
ELSE
	_HasMover	   := FALSE;
	ipCurrentMover := 0;
END_IF

IF _HasMover AND ipCurrentMover <> 0 THEN
	IF ipCurrentMover.std <> 0 THEN
		CASE _StationType OF
			E_StationType.Process:
				_StationReady := NOT ipCurrentMover.std.P_Busy;
			E_StationType.MultiMover:
				_StationReady := NOT ipCurrentMover.std.P_Busy AND (_MoverQueue.Count = _NumMoversRequired);
			E_StationType.DecisionPoint:
				_StationReady := _HasMover;
		END_CASE
	END_IF
END_IF

HMICommunication();
SUPER^.CyclicLogic();
END_METHOD

//! @summary Provides interlocks for HMI control and updates HMI status information for this component
METHOD PROTECTED HMICommunication

//! @description This method is called cyclically by <c>CyclicLogic()</c>
Station_HMI.Status.HasMover := _HasMover;
IF ipCurrentMover <> 0 THEN
	Station_HMI.Status.MoverID := ipCurrentMover.MoverBTN;
ELSE
	Station_HMI.Status.MoverID := '';
END_IF
END_METHOD

PROPERTY AllowQueing : BOOL
GET
AllowQueing := _AllowQueing;
END_GET
SET
_AllowQueing := AllowQueing;
END_SET
END_PROPERTY

PROPERTY CanReleaseMover : BOOL
SET
_CanReleaseMover := CanReleaseMover;
END_SET
END_PROPERTY

PROPERTY CurrentMover : I_XPlanarMover
GET
IF ipCurrentMover <> 0 THEN
	CurrentMover := ipCurrentMover;
END_IF
END_GET
END_PROPERTY

PROPERTY Error : BOOL
GET
Error := _Error;
END_GET
END_PROPERTY

METHOD Execute
VAR_INST
	i: UDINT := 1;
END_VAR
IF ipCurrentMover <> 0 THEN
	CASE StationState OF
		E_XplanarStationState.StationIdle: //Wait for mover to arrive in position
			IF _HasMover AND _StationReady AND NOT _StationComplete THEN
				IF ipCurrentMover.std <> 0 THEN
					IF (
					   ipTrackID <> 0 AND (ipCurrentMover.std.P_CommandMode = MC_PLANAR_MOVER_COMMAND_MODE.OnTrack OR ipCurrentMover.std.P_CommandMode = MC_PLANAR_MOVER_COMMAND_MODE.CRotationOnTrack)
					   	) OR (ipTrackID = 0 AND
					   (ipCurrentMover.std.P_CommandMode = MC_PLANAR_MOVER_COMMAND_MODE.FreeMovement OR ipCurrentMover.std.P_CommandMode = MC_PLANAR_MOVER_COMMAND_MODE.CRotationFreeMovement)) THEN
						StationState := E_XplanarStationState.ProcessMover;
					END_IF
				END_IF
			END_IF

		E_XplanarStationState.ProcessMover: //Perform the desired processes with the mover
			IF _StationComplete THEN
				IF _StationType = E_StationType.MultiMover THEN
					i := 1;
					StationState := E_XPlanarStationState.SendQueue;
				ELSE
					StationState := E_XplanarStationState.SquareUpMover;
				END_IF
			END_IF

		E_XplanarStationState.SquareUpMover: //Check mover for angle that allows X/Y Movement
			IF ipCurrentMover.std <> 0 THEN
				IF (ipCurrentMover.std.P_CommandMode = MC_PLANAR_MOVER_COMMAND_MODE.CRotationOnTrack) OR (ipCurrentMover.std.P_CommandMode = MC_PLANAR_MOVER_COMMAND_MODE.CRotationFreeMovement) THEN
					IF ipCurrentMover.SquareUp() THEN
						StationState := E_XplanarStationState.SendMoverAway;
					END_IF
				ELSE
					StationState := E_XplanarStationState.SendMoverAway;
				END_IF
			END_IF

		E_XplanarStationState.SendMoverAway: //Send the current lead mover away
			IF ipNextStation <> 0 AND _CanReleaseMover THEN
				IF (NOT ipNextStation.HasMover OR ipNextStation.AllowQueing) THEN
					IF ipCurrentMover.SendToStation(ipDestinationLocal := ipNextStation) THEN
						_MoverQueue.Dequeue();
						StationState := E_XplanarStationState.CycleComplete;
					END_IF
				END_IF
			END_IF
			
		E_XPlanarStationState.SendQueue:  //Send the mover queue away
			IF i <= _NumMoversRequired THEN
				IF   _MoverQueue.Queue[1].Destination <> 0 AND _MoverQueue.Queue[1].Destination.ID <> _ID THEN 
					IF _MoverQueue.Queue[1].SendToStation(ipDestinationLocal := _MoverQueue.Queue[1].Destination) THEN
						_MoverQueue.Dequeue();
						i := i + 1;
					END_IF
				ELSE
					IF _MoverQueue.Queue[1].SendToStation(ipDestinationLocal := ipNextStation) THEN
						_MoverQueue.Dequeue();
						i := i + 1;
					END_IF
				END_IF	
			ELSE
				i                       := 1;
				StationState := E_XplanarStationState.CycleComplete;
			END_IF

		E_XplanarStationState.CycleComplete: //Mover on its way out
			_StationReady := FALSE;
			StationState  := E_XplanarStationState.StationIdle;
	END_CASE
ELSE
	_StationComplete := FALSE;
	_StationReady	 := FALSE;
	StationState	 := E_XplanarStationState.StationIdle;
END_IF
END_METHOD

PROPERTY HasMover : BOOL
GET
HasMover := _HasMover;
END_GET
SET
_HasMover := HasMover;
END_SET
END_PROPERTY

PROPERTY ID : UDINT
GET
ID := _ID;
END_GET
SET
_ID := ID;
END_SET
END_PROPERTY

PROPERTY MoverQueue : REFERENCE TO FB_MoverQueue
GET
MoverQueue ref= _MoverQueue;
END_GET
END_PROPERTY

PROPERTY NextStation : I_XPlanarStation
GET
NextStation := ipNextStation;
END_GET
SET
ipNextStation := NextStation;
END_SET
END_PROPERTY

PROPERTY NumMoversRequired : UDINT
GET
NumMoversRequired := _NumMoversRequired;
END_GET
SET
_NumMoversRequired := NumMoversRequired;
END_SET
END_PROPERTY

PROPERTY Position : REFERENCE TO PositionXYC
GET
Position ref= _Position;
END_GET
END_PROPERTY

METHOD Recover : BOOL
VAR_INST
	TrackPos	 : LREAL;
	CorrectedPos : PositionXYC;
END_VAR

VAR
	Result : BOOL;
END_VAR
IF ipCurrentMover <> 0 THEN
	IF ipCurrentMover.std <> 0 THEN
		Recover := FALSE;
		CASE PrepState OF
			0: //Make sure there is a mover to recover
				IF _HasMover THEN
					ipCurrentMover.Destination := THIS^;
					IF ipCurrentMover.std.P_AtRotationPoint THEN
						PrepState := PrepState + 5;
					ELSE
						PrepState := PrepState + 10;
					END_IF
				ELSIF NOT _HasMover THEN
					Recover := TRUE;
				END_IF

			5: //SquareUP
				IF ipCurrentMover.SquareUp() THEN
					IF ipCurrentMover.Error THEN
						PrepState := 999;
					ELSE
						PrepState := PrepState + 5;
					END_IF
				END_IF

			10: //Check Mover Status
				CorrectedPos.SetValuesXYC(_Position.x, _Position.y, ipCurrentMover.std.P_ActPosition.c);
				IF ipCurrentMover.std.P_CommandMode = MC_PLANAR_MOVER_COMMAND_MODE.OnTrack THEN
					PrepState := PrepState + 40;
				ELSE
					PrepState := PrepState + 10;
				END_IF

			20: //Move to center of zone		
				Result := ipCurrentMover.std.MoveToPosition('InitMoverInStation',
															CorrectedPos,
															ipCurrentMover.MoveDynamics.Velo,
															ipCurrentMover.MoveDynamics.Accel,
															ipCurrentMover.MoveDynamics.Decel,
															ipCurrentMover.MoveDynamics.Jerk);

				PrepState := PrepState + 10;

			30: //Monitor Command Feedback
				IF ipCurrentMover.std.P_MoveToPosition.Done THEN
					PrepState := PrepState + 10;
				ELSIF ipCurrentMover.std.P_MoveToPosition.Error THEN
					_ErrorID  := ipCurrentMover.std.P_MoveToPosition.ErrorID;
					PrepState := 999;
				END_IF

			40: //If the station is configured on a track - Join mover
				IF ipTrackID <> 0 THEN
					IF ipCurrentMover.JoinTrack(ipTrackID) THEN
						IF ipCurrentMover.Error THEN
							PrepState := 999;
						ELSE
							PrepState := 100;
						END_IF
					END_IF
				ELSE
					PrepState := 90;
				END_IF

			50: //Mover to center of station
				IF ipTrackID <> 0 THEN
					IF ipTrackID.std <> 0 THEN
						TrackPos := ipTrackID.std.GetTrackPositionAt(CorrectedPos);
						Result	 := ipCurrentMover.std.MoveOnTrack('InitMoverInStation',
																   ipTrackID.std,
																   TrackPos,
																   ipCurrentMover.MoveDynamics.VeloSlow,
																   ipCurrentMover.MoveDynamics.Accel,
																   ipCurrentMover.MoveDynamics.Jerk,
																   ipCurrentMover.MoveDynamics.Gap,
																   Tc3_Mc3PlanarMotion.MC_DIRECTION.mcDirectionShortestWay);

						PrepState := PrepState + 10;
					ELSE ///Marc TODO:  this is extra just checking the pointers how to handle?
						_ErrorID  := 16#FFFF;
						PrepState := 999;
					END_IF
				ELSE
					_ErrorID  := 16#FFFF;
					PrepState := 999;
				END_IF

			60: //Monitor Command Feedback
				IF ipCurrentMover.std.P_MoveOnTrack.Done THEN
					PrepState := 100;
				ELSIF ipCurrentMover.std.P_MoveOnTrack.Error THEN
					_ErrorID  := ipCurrentMover.std.P_MoveOnTrack.ErrorID;
					PrepState := 999;
				END_IF

			100: //Monitor Command feedback
				Recover	  := TRUE;
				PrepState := 0;

			999: //Error
				_Error	 := TRUE;
				_ErrorID := ipCurrentMover.ErrorID;
		END_CASE
	ELSE //No Mover to Initialize with the Standard library
		Recover	  := TRUE;
		PrepState := 0;
	END_IF
ELSE //No Mover to Initialize
	Recover	  := TRUE;
	PrepState := 0;
END_IF
END_METHOD

METHOD Reset : BOOL
StationState := E_XplanarStationState.StationIdle;
PrepState	 := 0;
_Error		 := FALSE;
Reset		 := true;
END_METHOD

PROPERTY Size : REFERENCE TO Position2D_LREAL
GET
Size ref= _Size;
END_GET
END_PROPERTY

PROPERTY StationComplete : BOOL
SET
_StationComplete := StationComplete;
END_SET
END_PROPERTY

PROPERTY StationReady : BOOL
GET
StationReady := _StationReady;
END_GET
END_PROPERTY

PROPERTY StationType : E_StationType
GET
StationType := _StationType;
END_GET
SET
_StationType := StationType;
END_SET
END_PROPERTY

PROPERTY TrackID : I_XPlanarTrack
GET
TrackID := ipTrackID;
END_GET
SET
ipTrackID := TrackID;
END_SET
END_PROPERTY

END_FUNCTION_BLOCK

// Track/FB_XPlanarTrackSegment
FUNCTION_BLOCK FB_XPlanarTrackSegment IMPLEMENTS I_XPlanarTrack
VAR
	TrackStandard : FB_TrackStandard;
	_TrackLength  : LREAL;
	_Error		  : BOOL;
	_TrackTable	  : FB_TrackTable;
	_TrackID	  : UDINT;
	_ErrorID	  : UDINT;
	_ErrorInfo	  : STRING;
	BuildState	  :
		(Init,
		CheckTrackTable,
		BuildTrackSegment,
		MonitorBuildFeedback,
		BuildComplete,
		BuildError);
	Track_HMI : ST_Track_HMI;
END_VAR

METHOD Clear : BOOL
VAR_INST
	nStateReset : UINT;
END_VAR
Clear := FALSE;
CASE nStateReset OF
	0:
		nStateReset := 10;

	10:
		IF TrackStandard.P_State = MC_PLANAR_STATE.Error OR TrackStandard.P_State = MC_PLANAR_STATE.ErrorPending THEN
			nStateReset := nStateReset + 1;
		ELSE
			nStateReset := nStateReset + 10;
		END_IF

	11:
		IF TrackStandard.Reset() THEN
			nStateReset := nStateReset + 1;
		END_IF

	12:
		IF TrackStandard.P_Reset.Done THEN
			nStateReset := nStateReset + 8;
		END_IF

	20:
		_ErrorInfo	:= '';
		_Error		:= FALSE;
		nStateReset := 10;
		Clear		:= TRUE;
		nStateReset := 0;
END_CASE
END_METHOD

PROPERTY Error : BOOL
GET
Error := _Error;
END_GET
END_PROPERTY

PROPERTY ErrorInfo : STRING
GET
ErrorInfo := _ErrorInfo;
END_GET
END_PROPERTY

PROPERTY ID : UDINT
GET
ID := _TrackID;
END_GET
SET
_TrackID := ID;
END_SET
END_PROPERTY

PROPERTY MoverCount : UDINT
GET
MoverCount := TrackStandard.stTrackRef.MCTOPLC_STD.MoverCountOnTrack;
END_GET
END_PROPERTY

PROPERTY OpMode : MC_PLANAR_TRACK_OPERATION_MODE
GET
OpMode := TrackStandard.stTrackRef.MCTOPLC_STD.OperationMode;
END_GET
END_PROPERTY

PROPERTY std : I_TrackStandard
GET
std := TrackStandard;
END_GET
END_PROPERTY

PROPERTY TrackLength : LREAL
GET
TrackLength := _TrackLength;
END_GET
END_PROPERTY

PROPERTY TrackTable : REFERENCE TO FB_TrackTable
GET
TrackTable ref= _TrackTable;
END_GET
END_PROPERTY

METHOD Build : BOOL
VAR_INST
	sIndexWhereTheCheckFailed : UINT;
	TrackTableTemp			  : ARRAY[1..Tc3_XPlanarStandard.maxNumTrackPoints] OF ST_TrackTable;
END_VAR
Build := FALSE;
CASE BuildState OF
	Init: // Starting with an empty table. 
		BuildState := CheckTrackTable;

	CheckTrackTable: // Checking the track table for plausibility
		IF _TrackTable.CheckTrackTable() <> 0 THEN
			IF _TrackTable.P_TrackTableCheckResult THEN
				BuildState := BuildTrackSegment; // Plausibility test succeeded.
			ELSE
				_ErrorInfo				  := _TrackTable.P_InfoText;
				sIndexWhereTheCheckFailed := _TrackTable.P_TrackCheckImplausibleTableIndex;
				TrackTableTemp			  := _TrackTable.P_Table;
				BuildState				  := BuildError;
			END_IF
		END_IF

	BuildTrackSegment: // Building the track	
		IF TrackStandard.BuildTrackExt(_TrackTable) THEN
			BuildState := MonitorBuildFeedback;
		END_IF

	MonitorBuildFeedback: //Monitor Track Build Feedback
		IF TrackStandard.P_BuildTrackExt.Done THEN
			BuildState := BuildComplete;
		ELSIF TrackStandard.P_BuildTrackExt.Error THEN
			BuildState := BuildError;
		END_IF

	BuildComplete: // Track build done
		_TrackLength := TrackStandard.GetLength();
		Build		 := TRUE;

	BuildError: //Error

		// In case of failed plausibility test check the creation of the above track table.

		// A Line must always begin with E_PointType.Line_Start and end with E_PointType.Line_End.

		// A Circle must always be added in the order E_PointType.Circle_Start, E_PointType.Circle_Center, E_PointType.Circle_End.

		// Check the info text for further information:	
		_ErrorID   := TrackStandard.P_BuildTrackExt.ErrorID;
		_ErrorInfo := TrackStandard.P_BuildTrackExtInfoText;
		_Error	   := TRUE;
END_CASE
END_METHOD

METHOD CyclicLogic
VAR_INPUT
END_VAR

VAR
	Result : BOOL;
END_VAR
Result	   := TrackStandard.Cycle();
_ErrorInfo := TrackStandard.P_BuildTrackExtInfoText;
END_METHOD

METHOD HMICommunication
VAR_INPUT
END_VAR
Track_HMI.Status.State := TrackStandard.stTrackRef.MCTOPLC_STD.State;
;
Track_HMI.Status.OperationMode	  := TrackStandard.stTrackRef.MCTOPLC_STD.OperationMode;
Track_HMI.Status.CalculatedLength := _TrackLength;
Track_HMI.Status.MoverCount		  := TrackStandard.stTrackRef.MCTOPLC_STD.MoverCountOnTrack;
END_METHOD

END_FUNCTION_BLOCK

// FB_Component_XPlanar
FUNCTION_BLOCK FB_Component_XPlanar EXTENDS FB_ComponentBase
VAR
	XPlanarSystem	  : FB_XPlanarSystem;
	HaltDynamics	  : ST_HaltDynamics;
	_Movers			  : ARRAY[1..Tc3_XPlanarStandard.Params_XPlanar.moverCount] OF FB_XPlanarMover;
	_Tracks			  : ARRAY[1..Tc3_XPlanarStandard.Params_XPlanar.maxTrackCount] OF FB_XPlanarTrackSegment;
	XPlanarBaseAlarms : ARRAY[1..XPLANAR_BASE_ALARM_COUNT] OF FB_TcAlarm;

	//HMI
	XPlanar_HMI : ST_Xplanar_HMI;
	Force		: Force6D;

	//Helper Vars
	_TracksInitialized	: BOOL;
	_TileCount			: UDINT;
	OpMode				: OperationMode;
	SimType				: MoverType;
	AbortState			: UDINT;
	TrackBuildState		: UDINT;
	CheckMoverState		: UDINT;
	CheckTilePowerState : UDINT;
	EnableGroupState	: UDINT;
	EnableMoversState	: UDINT;
	EnableTrackState	: UDINT;
	RedetectState		: UDINT;
	ResetState			: UDINT;
END_VAR

VAR CONSTANT
	XPLANAR_BASE_ALARM_COUNT : UINT := 6; // Number of defined events configured in the tmc file
END_VAR

//! @summary Initializes event function blocks using this components's name
{attribute 'call_after_online_change_slot' := '<slot>'}
METHOD PROTECTED CreateEvents

//! @description This method is called by <c>Initialize()</c> as required
F_CreateAllEventsInClass(Alarms		:= XPlanarBaseAlarms,
						 ClassSize	:= SIZEOF(TC_EVENTS.XPlanarBase),
						 pInitEvent := ADR(TC_EVENTS.XPlanarBase.InitReferenceEvent),
						 Prefix		:= Name);

SUPER^.CreateEvents();
END_METHOD

//! @summary Provides interlocks for HMI control and updates HMI status information for this component
METHOD PROTECTED HMICommunication

//! @description This method is called cyclically by <c>CyclicLogic()</c>
SUPER^.HMICommunication();
XPlanar_HMI.Status.Initialized		:= _TracksInitialized;
XPlanar_HMI.Status.NumberOfMovers	:= Tc3_XPlanarStandard.Params_XPlanar.moverCount;
XPlanar_HMI.Status.NumberOfStations := Tc3_XPlanarStandard.Params_XPlanar.maxNumStation;
XPlanar_HMI.Status.NumberOfTracks	:= Tc3_XPlanarStandard.Params_XPlanar.maxTrackCount;

///XPlanar_HMI.Status.PowerOK := XPlanarSystem.
XPlanar_HMI.Status.TileCount := _TileCount;
END_METHOD

//! Provides basic error detection and event handling for this component
METHOD PROTECTED Monitoring
(*! @descriptionThis method is called cyclically by <c>CyclicLogic()</c>*)
VAR
	i	   : UDINT;
	Result : HRESULT;
END_VAR
FOR i := 1 TO Tc3_XPlanarStandard.Params_XPlanar.moverCount DO
	IF _Movers[i].std.P_State = MC_PLANAR_STATE.Error AND NOT XPlanarBaseAlarms[E_XPlanarBase.MoverError].bRaised THEN
		RaiseAlarmWithStrings(Alarm := XPlanarBaseAlarms[E_XPlanarBase.MoverError], CONCAT('Mover ', _Movers[i].MoverBTN), 'Faulted');
	ELSIF NOT _Movers[i].std.P_State = MC_PLANAR_STATE.Error AND XPlanarBaseAlarms[E_XPlanarBase.MoverError].bRaised THEN
		Result := XPlanarBaseAlarms[E_XPlanarBase.MoverError].Clear(0, 0);
	END_IF

	IF _Movers[i].Error AND NOT XPlanarBaseAlarms[E_XPlanarBase.CommandError].bRaised THEN
		RaiseAlarmWithStrings(Alarm := XPlanarBaseAlarms[E_XPlanarBase.CommandError], CONCAT('Mover ', _Movers[i].MoverBTN), CONCAT(_Movers[i].ErrorInfo, TO_STRING(_Movers[i].ErrorID)));
	ELSIF NOT _Movers[i].Error AND XPlanarBaseAlarms[E_XPlanarBase.CommandError].bRaised THEN
		Result := XPlanarBaseAlarms[E_XPlanarBase.CommandError].Clear(0, 0);
	END_IF
END_FOR

//Catch the XPlanar errors
_CurrentAlarmSeverity := F_GetMaxSeverityRaised(Alarms := XPlanarBaseAlarms, CurrentSeverity := _CurrentAlarmSeverity);
END_METHOD

//! @summary This method serves as the entry point for all underlying FB logic
METHOD PUBLIC CyclicLogic
//! @description This method should be called cyclically by descendant function blocks by invoking <c>SUPER^.CyclicLogic()</c>.  Alternatively, the contents of this method could be reimplemented entirely in which case a call to this method would not be necessary.
VAR_Inst
	i			 : UDINT;
	IoIdx		 : UINT;
	GetMoverInfo : BOOL;
END_VAR

VAR
	ipResultMover : I_XPlanarMoverStandard;
	ResultTrack	  : BOOL;
END_VAR
//Update Xplanar system status
XPlanarSystem.Cycle();

//Update Mover status
FOR i := 1 TO Tc3_XPlanarStandard.Params_XPlanar.moverCount DO
	ipResultMover := XPlanarSystem.SetMoverStandard(i, _Movers[i].std);
	_Movers[i].CyclicLogic();
END_FOR

//Update Track status 
FOR i := 1 TO Tc3_XPlanarStandard.Params_XPlanar.maxTrackCount DO
	ResultTrack	  := XPlanarSystem.SetTrackStandard(i, _Tracks[i].std);
	_Tracks[i].ID := i;
	_Tracks[i].CyclicLogic();
END_FOR

//Update Station IDs
FOR i := 1 TO Tc3_XPlanarStandard.Params_XPlanar.maxNumStation DO
	IF ip.Stations[i] <> 0 THEN
		ip.Stations[i].ID := i;
	END_IF
END_FOR

//Make sure things are initialized
IF NOT _InitComplete THEN
	_InitComplete := Initialize();
END_IF

SUPER^.CyclicLogic();
END_METHOD

METHOD Abort : BOOL
VAR
	i	   : UDINT := 1;
	Result : BOOL;
END_VAR
VAR_INST
	ErrString : STRING;
END_VAR
Abort := FALSE;
CASE AbortState OF
	0:
		AbortState := AbortState + 10;

	10: //Halt System
		IF XPlanarSystem.HaltSystem() THEN
			AbortState := AbortState + 10;
		END_IF
	
	20: //Monitor Halt System Feedback
		IF XPlanarSystem.P_HaltSystem.Done THEN
			AbortState := AbortState + 10;
		ELSIF XPlanarSystem.P_HaltSystem.Error THEN
			ErrString := 'Error Halting System';
			AbortState := 999;
		END_IF

	30: //Disable Movers
		IF XPlanarSystem.DisableMovers() THEN
			AbortState := AbortState + 10;
		END_IF

	40: //Check disable command feedback
		IF XPlanarSystem.P_DisableMovers.Done THEN
			AbortState := AbortState + 10;
		ELSIF XPlanarSystem.P_DisableMovers.Error THEN
			ErrString := 'NotAll Movers Disabled';
			AbortState := 999;
		END_IF

	50: //Cleanup mover command states
		FOR i := 1 TO Tc3_XPlanarStandard.Params_XPlanar.moverCount DO
			Result := _Movers[i].ClearCmd();
		END_FOR
		
		AbortState := AbortState + 10;

	60: //Disable Tracks
		IF XPlanarSystem.DisableTracks() THEN
			AbortState := AbortState + 10;
		END_IF

	70: //Monitor track disable feedback
		IF XPlanarSystem.P_DisableTracks.Done THEN
			AbortState := AbortState + 10;
		ELSIF XPlanarSystem.P_DisableTracks.Error THEN
			ErrString := 'NotAll Tracks Disabled';
			AbortState := 999;
		END_IF

	80: //Make sure sequences are reset
		TrackBuildState		:= 0;
		CheckMoverState		:= 0;
		CheckTilePowerState := 0;
		EnableGroupState	:= 0;
		EnableMoversState	:= 0;
		EnableTrackState	:= 0;
		RedetectState		:= 0;
		ResetState			:= 0;
		AbortState			:= AbortState + 10;

	90: //Abort Complete	
		Abort	   := TRUE;
		AbortState := 0;

	999: //Error
		Abort	   := TRUE;
		AbortState := 0;
		_Error	   := TRUE;
		RaiseAlarmWithStrings(Alarm := XPlanarBaseAlarms[E_XPlanarBase.SystemError], 'AbortingError', ErrString);
END_CASE
END_METHOD

METHOD BuildTracks : BOOL
VAR_INST
	TrackToInit : UDINT := 1;
END_VAR

VAR
	Result : DINT;
END_VAR
BuildTracks := FALSE;
CASE TrackBuildState OF
	0: //Init
		IF _TracksInitialized THEN
			TrackBuildState := 30;
		ELSE
			TrackToInit		:= 1;
			TrackBuildState := TrackBuildState + 10;
		END_IF

	10: //Clear any existing Track Data
		IF _Tracks[TrackToInit].Clear() THEN
			TrackBuildState := TrackBuildState + 10;
		END_IF

	20: //Build the Track Segment
		IF NOT _Tracks[TrackToInit].Error THEN
			IF _Tracks[TrackToInit].Build() THEN
				Result := ADSLOGSTR(ADSLOG_MSGTYPE_HINT, 'Track Segment %s ', CONCAT(TO_STRING(TrackToInit), ' Build Success'));
				IF TrackToInit >= Tc3_XPlanarStandard.Params_XPlanar.maxTrackCount THEN
					TrackBuildState := TrackBuildState + 10;
				ELSE
					TrackToInit		:= TrackToInit + 1;
					TrackBuildState := 10;
				END_IF
			END_IF
		ELSE
			TrackBuildState := 999;
		END_IF

	30: //Track Build Complete
		_TracksInitialized := TRUE;
		BuildTracks		   := TRUE;
		TrackBuildState	   := 0;

	999: //Error State
		RaiseAlarmWithStrings(Alarm := XPlanarBaseAlarms[E_XPlanarBase.TrackError], CONCAT('Segment ', TO_STRING(_Tracks[TrackToInit].ID)), _Tracks[TrackToInit].ErrorInfo);
		_Error			:= TRUE;
		TrackBuildState := 0;
		BuildTracks		:= TRUE;
END_CASE
END_METHOD

METHOD CheckMovers : BOOL
CheckMovers := FALSE;
CASE CheckMoverState OF
	0: //Init
		_Error			:= FALSE;
		CheckMoverState := CheckMoverState + 10;

	10: //Check for lost movers
		IF XPlanarSystem.CheckValidMovers() THEN
			CheckMoverState := CheckMoverState + 10;
		END_IF

	20: //Monitor Command Feedback
		IF XPlanarSystem.P_CheckValidMovers.bDone THEN
			IF XPlanarSystem.P_CheckValidMovers.bMoverLost THEN
				CheckMoverState := 999;
			ELSE
				CheckMoverState := CheckMoverState + 10;
			END_IF
		END_IF

	30: //Mover Check OK
		CheckMovers		:= TRUE;
		CheckMoverState := 0;

	999: //Lost Mover detected
		RaiseAlarmWithStrings(Alarm := XPlanarBaseAlarms[E_XPlanarBase.SystemError], 'Not all movers present', 'Lost Mover Possible');
		_Error			:= TRUE;
		CheckMoverState := 0;
		CheckMovers		:= TRUE;
END_CASE
END_METHOD

METHOD CheckTilePower : BOOL
VAR_INST
	TileCount : UDINT;
END_VAR

VAR
	PowerOK : BOOL;
	i		: UINT;
	Result	: BOOL;
END_VAR
CheckTilePower := FALSE;
IF XPlanarSystem.ipDriver <> 0 THEN
	CASE CheckTilePowerState OF
		0: //Init -Check Operation Mode
			_Error	 := FALSE;
			_ErrorID := 0;
			IF XPlanarSystem.ipDriver.XpuTcIo(1).GetOperationMode() = 0 THEN
				CheckTilePowerState := CheckTilePowerState + 10;
			ELSE
				CheckTilePowerState := 30;
			END_IF

		10: //Get Tile Count
			TileCount			:= XPlanarSystem.ipDriver.XpuTcIo(1).GetTileCount();
			CheckTilePowerState := CheckTilePowerState + 10;

		20: //Check DC Link of each tile
			PowerOK := TRUE;
			FOR i := 1 TO UDINT_TO_UINT(TileCount) DO
				IF XPlanarSystem.ipDriver.XpuTcIo(1).TileCoE(1, i).DiagData <> 0 THEN
					Result	:= XPlanarSystem.ipDriver.XpuTcIo(1).TileCoE(1, i).DiagData.Update();
					PowerOK := PowerOK AND XPlanarSystem.ipDriver.XpuTcIo(1).TileCoE(1, i).DiagData.DcLinkOk;
				ELSE ///Marc TODO: how do we handle this?  Maybe nothing??
					;
				END_IF
			END_FOR

			IF PowerOK THEN
				CheckTilePowerState := CheckTilePowerState + 10;
			ELSE
				CheckTilePowerState := 999;
			END_IF

		30: // DC LinkOK
			CheckTilePower		:= TRUE;
			CheckTilePowerState := 0;

		999: //DC LinkNot OK
			RaiseAlarmWithStrings(Alarm := XPlanarBaseAlarms[E_XPlanarBase.TileError], 'TilePowerNotOK', 'CheckPowerConnections');
			_Error				:= TRUE;
			CheckTilePower		:= TRUE;
			CheckTilePowerState := 0;
	END_CASE
ELSE ///Marc TODO:  how to handle this Maybe do nothing
	;
END_IF
END_METHOD

METHOD EnableGroup : BOOL
EnableGroup := FALSE;
CASE EnableGroupState OF
	0:
		EnableGroupState := EnableGroupState + 10;

	10: //Enable the group
		IF XPlanarSystem.EnableGroup() THEN
			EnableGroupState := EnableGroupState + 10;
		END_IF

	20: //Monitor Command Feedback
		IF XPlanarSystem.P_EnableGroup.Done THEN
			EnableGroupState := EnableGroupState + 10;
		ELSIF XPlanarSystem.P_EnableGroup.Error THEN
			RaiseAlarmWithStrings(Alarm := XPlanarBaseAlarms[E_XPlanarBase.SystemError], 'EnableGroupError', TO_STRING(XPlanarSystem.P_EnableGroup.ErrorID));
			EnableGroupState := 999;
		END_IF

	30: //Add Xplanar Environment to Group
		IF XPlanarSystem.AddEnvironmentToGroup() THEN
			EnableGroupState := EnableGroupState + 10;
		END_IF

	40: //Monitor Command Feedback
		IF XPlanarSystem.P_AddEnviromentToGroup.Done THEN
			EnableGroupState := EnableGroupState + 10;
		ELSIF XPlanarSystem.P_AddEnviromentToGroup.Error THEN
			RaiseAlarmWithStrings(Alarm := XPlanarBaseAlarms[E_XPlanarBase.SystemError], 'AddEnvironmentError', TO_STRING(XPlanarSystem.P_AddEnviromentToGroup.ErrorID));
			EnableGroupState := 999;
		END_IF

	50: //Enabling Complete
		EnableGroupState := 0;
		EnableGroup		 := TRUE;

	999: //Error Enabling Group
		_Error		:= TRUE;
		EnableGroup := TRUE;
END_CASE
END_METHOD

METHOD EnableMovers : BOOL
VAR_INPUT
	UseGroup : BOOL;
END_VAR

VAR_INST
	i : UINT := 1;
END_VAR
EnableMovers := FALSE;
CASE EnableMoversState OF
	0: //Init
		i				  := 1;
		EnableMoversState := EnableMoversState + 10;

	10: //Enable Movers
		IF i <= Tc3_XPlanarStandard.Params_XPlanar.moverCount THEN
			_Movers[i].IODriver := XPlanarSystem.ipDriver.XpuTcIo(1).MoverTcIo(i);
			IF _Movers[i].Enable() THEN
				IF NOT _Movers[i].Error THEN
					i := i + 1;
				ELSE
					_ErrorID		  := _Movers[i].ErrorID;
					EnableMoversState := 999;
				END_IF
			END_IF
		ELSE
			i := 1;
			IF UseGroup THEN
				EnableMoversState := EnableMoversState + 10;
			ELSE
				EnableMoversState := 40;
			END_IF
		END_IF

	20: //Add Movers to Group
		IF XPlanarSystem.AddMoversToGroup() THEN
			EnableMoversState := EnableMoversState + 10;
		END_IF

	30: //Monitor Command Feedback
		IF XPlanarSystem.P_AddMoversToGroup.Done THEN
			EnableMoversState := EnableMoversState + 10;
		ELSIF XPlanarSystem.P_AddMoversToGroup.Error THEN
			_ErrorID		  := XPlanarSystem.P_AddEnviromentToGroup.ErrorID;
			EnableMoversState := 999;
		END_IF

	40: //Enable Movers Complete
		EnableMoversState := 0;
		EnableMovers	  := TRUE;

	999: //Error Enabling Movers
		EnableMoversState := 0;
		EnableMovers	  := TRUE;
		_Error			  := TRUE;
		RaiseAlarmWithStrings(Alarm := XPlanarBaseAlarms[E_XPlanarBase.SystemError], CONCAT('Mover ', TO_STRING(i)), CONCAT('EnableError ', TO_STRING(_ErrorID)));
END_CASE
END_METHOD

METHOD EnableTracks : BOOL
VAR_INPUT
	UseGroup : BOOL;
END_VAR

VAR_INST
	i : UDINT := 1;
END_VAR

VAR
	Result : BOOL;
END_VAR
EnableTracks := FALSE;
CASE EnableTrackState OF
	0:
		i				 := 1;
		EnableTrackState := EnableTrackState + 10;

	10: //Enable Track Seqment
		IF i <= Tc3_XPlanarStandard.Params_XPlanar.maxTrackCount THEN
			IF _Tracks[i].std.P_State <> MC_PLANAR_STATE.Enabled THEN
				IF _Tracks[i].std <> 0 THEN
					Result := _Tracks[i].std.Enable();
				ELSE
					EnableTrackState := 10000;
				END_IF
			END_IF

			EnableTrackState := EnableTrackState + 1;
		ELSE
			i := 1;
			IF UseGroup THEN
				EnableTrackState := EnableTrackState + 10;
			ELSE
				EnableTrackState := 40;
			END_IF
		END_IF

	11: //Monitor Command Feedback
		IF _Tracks[i].std <> 0 THEN
			IF _Tracks[i].std.P_Enable.Done OR _Tracks[1].OpMode = MC_PLANAR_TRACK_OPERATION_MODE.Standing THEN
				i				 := i + 1;
				EnableTrackState := 10;
			ELSIF _Tracks[i].std.P_Enable.Error THEN
				EnableTrackState := 999;
			END_IF
		ELSE
			EnableTrackState := 10000;
		END_IF

	20: //Add Tracks to Group
		IF XPlanarSystem.AddTracksToGroup() THEN
			EnableTrackState := EnableTrackState + 10;
		END_IF

	30: //Monitor Command Feedback
		IF XPlanarSystem.P_AddTracksToGroup.Done THEN
			EnableTrackState := EnableTrackState + 10;
		ELSIF XPlanarSystem.P_AddTracksToGroup.Error THEN
			EnableTrackState := 999;
		END_IF

	40: //Enable Tracks Complete
		EnableTrackState := 0;
		EnableTracks	 := TRUE;

	999: //Error Enabling Track Segments
		EnableTrackState := 0;
		EnableTracks	 := TRUE;
		_Error			 := TRUE;
		RaiseAlarmWithStrings(Alarm := XPlanarBaseAlarms[E_XPlanarBase.TrackError], CONCAT('Track ', TO_STRING(i)), CONCAT('EnableError ', TO_STRING(_Tracks[i].std.P_Enable.ErrorID)));

	10000:
		; ///Marc TODO: do we need to handle this?  Should never happen.
END_CASE
END_METHOD

//! @summary Basic component initialization logic
METHOD PROTECTED Initialize : BOOL;
//! @description This method is called by <c>CyclicLogic()</c> as required
VAR_INST
	i			  : UDINT;
	SequenceState : UDINT;
	TrackToInit	  : UDINT := 1;
END_VAR
Initialize := FALSE;
CASE SequenceState OF
	0: //Init
		IF SUPER^.Initialize() THEN
			SequenceState := SequenceState + 10;
		END_IF

	10: //Set Mover references
		FOR i := 1 TO Tc3_XPlanarStandard.Params_XPlanar.moverCount DO
			_Movers[i].MoverIndex := i;
			ip.Movers[i]		  := _Movers[i];
		END_FOR

		FOR i := 1 TO Tc3_XPlanarStandard.Params_XPlanar.maxTrackCount DO
			ip.Tracks[i] := _Tracks[i];
		END_FOR

		SequenceState := SequenceState + 10;

	20: //Set Mover Halt Dynamics
		HaltDynamics.Mode				  := E_HaltDynamicsMode.AxisX_AxisY_CoordinatedOnPath;
		HaltDynamics.PathXY.fVelocity	  := 500.0;
		HaltDynamics.PathXY.fAcceleration := 10000.0;
		HaltDynamics.PathXY.fDeceleration := 10000.0;
		HaltDynamics.PathXY.fJerk		  := 100000.0;
		HaltDynamics.AxisA.fVelocity	  := 10.0;
		HaltDynamics.AxisA.fAcceleration  := 100.0;
		HaltDynamics.AxisA.fDeceleration  := 100.0;
		HaltDynamics.AxisA.fJerk		  := 100.0;
		HaltDynamics.AxisB.fVelocity	  := 10.0;
		HaltDynamics.AxisB.fAcceleration  := 100.0;
		HaltDynamics.AxisB.fDeceleration  := 100.0;
		HaltDynamics.AxisB.fJerk		  := 100.0;
		HaltDynamics.AxisC.fVelocity	  := 36.0;
		HaltDynamics.AxisC.fAcceleration  := 360.0;
		HaltDynamics.AxisC.fDeceleration  := 360.0;
		HaltDynamics.AxisC.fJerk		  := 360.0;
		FOR i := 1 TO Tc3_XPlanarStandard.Params_XPlanar.moverCount DO
			_Movers[i].std.P_HaltDynamics := HaltDynamics;
		END_FOR

		SequenceState := SequenceState + 10;

	30: //Init Complete
		Initialize := TRUE;

	999: // Init Error
END_CASE
END_METHOD

METHOD MoverRedetect : BOOL
VAR_INST
	MoverDetectionInfo : ST_TcIoMoverDetectionInfos;
END_VAR

VAR
	Result : BOOL;
END_VAR
MoverRedetect := FALSE;
CASE RedetectState OF
	0: //Init
		RedetectState := RedetectState + 10;

	10: //Start Mover Detection
		IF XPlanarSystem.ipDriver <> 0 THEN
			Result		  := XPlanarSystem.ipDriver.XpuTcIo(1).SetStartMoverRedetection();
			RedetectState := RedetectState + 10;
		ELSE
			; ///Marc TODO: How to handle? Maybe never.
		END_IF

	20: //Get detection feedback
		IF XPlanarSystem.ipDriver <> 0 THEN
			MoverDetectionInfo := XPlanarSystem.ipDriver.XpuTcIo(1).GetMoverDetectionInfos();
			RedetectState	   := RedetectState + 10;
		ELSE
			; ///Marc TODO: How to handle? Maybe never.
		END_IF

	30: //Evaluate detection results
		IF MoverDetectionInfo.TotalExpected <> MoverDetectionInfo.TotalDetected THEN
			RaiseAlarmWithStrings(Alarm := XPlanarBaseAlarms[E_XPlanarBase.SystemError], 'MoverCountInvald', 'Not all Movers Detected');
		END_IF

		RedetectState := RedetectState + 1;

	31:
		IF MoverDetectionInfo.APM4220Expected <> MoverDetectionInfo.APM4220Detected THEN
			RaiseAlarmWithStrings(Alarm := XPlanarBaseAlarms[E_XPlanarBase.SystemError], 'MoverCountInvald', 'Not all AMP4220 Detected');
		END_IF

		RedetectState := RedetectState + 1;

	32:
		IF MoverDetectionInfo.APM4221Expected <> MoverDetectionInfo.APM4221Detected THEN
			RaiseAlarmWithStrings(Alarm := XPlanarBaseAlarms[E_XPlanarBase.SystemError], 'MoverCountInvald', 'Not all AMP4221 Detected');
		END_IF

		RedetectState := RedetectState + 1;

	33:
		IF MoverDetectionInfo.APM4330Expected <> MoverDetectionInfo.APM4330Detected THEN
			RaiseAlarmWithStrings(Alarm := XPlanarBaseAlarms[E_XPlanarBase.SystemError], 'MoverCountInvald', 'Not all AMP4330 Detected');
		END_IF

		RedetectState := RedetectState + 1;

	34:
		IF MoverDetectionInfo.APM4550Expected <> MoverDetectionInfo.APM4550Detected THEN
			RaiseAlarmWithStrings(Alarm := XPlanarBaseAlarms[E_XPlanarBase.SystemError], 'MoverCountInvald', 'Not all AMP4550 Detected');
		END_IF

		RedetectState := 40;

	40: //Mover detection complete
		MoverRedetect := TRUE;
		RedetectState := 0;
END_CASE
END_METHOD

METHOD RecoverStations : BOOL
VAR_INST
	RecoverIndex : UDINT := 1;
END_VAR
RecoverStations := FALSE;
IF RecoverIndex <= Tc3_XPlanarStandard.Params_XPlanar.maxNumStation THEN
	IF ip.Stations[RecoverIndex].Recover() THEN
		RecoverIndex := RecoverIndex + 1;
	END_IF
ELSE
	RecoverStations := TRUE;
	RecoverIndex	:= 1;
END_IF
END_METHOD

//! @summary Clears error flags and error IDs for this component
METHOD PUBLIC Reset : BOOL
VAR
	i : UDINT;
END_VAR
Reset := FALSE;
CASE ResetState OF
	0:
		i		   := 1;
		ResetState := ResetState + 10;

	10: //Reset Movers
		IF XPlanarSystem.ResetMovers() THEN
			ResetState := ResetState + 10;
		END_IF

	20: //Monitor Mover Reset Feedback
		IF XPlanarSystem.P_ResetMovers.Done THEN
			ResetState := ResetState + 10;
		ELSIF XPlanarSystem.P_ResetMovers.Error THEN
			RaiseAlarmWithStrings(Alarm := XPlanarBaseAlarms[E_XPlanarBase.SystemError], 'MoverResetError', TO_STRING(XPlanarSystem.P_ResetMovers.ErrorID));
			ResetState := 999;
		END_IF

	30: //Reset Tracks
		IF XplanarSystem.ResetTracks() THEN
			ResetState := ResetState + 10;
		END_IF

	40: //Monitor Track Reset Feedback
		IF XPlanarSystem.P_ResetTracks.Done THEN
			ResetState := ResetState + 10;
		ELSIF XPlanarSystem.P_ResetTracks.Error THEN
			RaiseAlarmWithStrings(Alarm := XPlanarBaseAlarms[E_XPlanarBase.SystemError], 'TrackResetError', TO_STRING(XPlanarSystem.P_ResetTracks.ErrorID));
			ResetState := 999;
		END_IF

	50: //System Prep Complete
		F_ClearAllEventsInClass(XPlanarBaseAlarms);
		IF SUPER^.Reset() THEN
			ResetState := 0;
			Reset	   := TRUE;
		END_IF

		ResetState := 0;
		_Error	   := FALSE;
		Reset	   := TRUE;

	999: //Error Enabling Track Segments
		_Error	   := TRUE;
		ResetState := 0;
END_CASE
END_METHOD

PROPERTY TileCount : UDINT
GET
IF XPlanarSystem.ipDriver <> 0 THEN
	IF XPlanarSystem.ipDriver.XpuTcIo(1).GetOperationMode() = 0 THEN
		TileCount := XPlanarSystem.ipDriver.XpuTcIo(1).GetTileCount();
	END_IF
ELSE
	TileCount := 0; ///Marc TODO: What to return if the interface is not good?
END_IF
END_GET
END_PROPERTY

PROPERTY TracksInitialized : BOOL
GET
TracksInitialized := _TracksInitialized;
END_GET
END_PROPERTY

PROPERTY Xpu : I_TcIoXPlanarProcessingUnit
GET
IF XPlanarSystem.ipDriver <> 0 THEN
	Xpu := XPlanarSystem.ipDriver.XpuTcIo(1);
ELSE
	Xpu := 0; ///Marc TODO:  is zero ok to return?
END_IF
END_GET
END_PROPERTY

END_FUNCTION_BLOCK
